// ---- VISUs/Tela_Manual_1.TcVIS
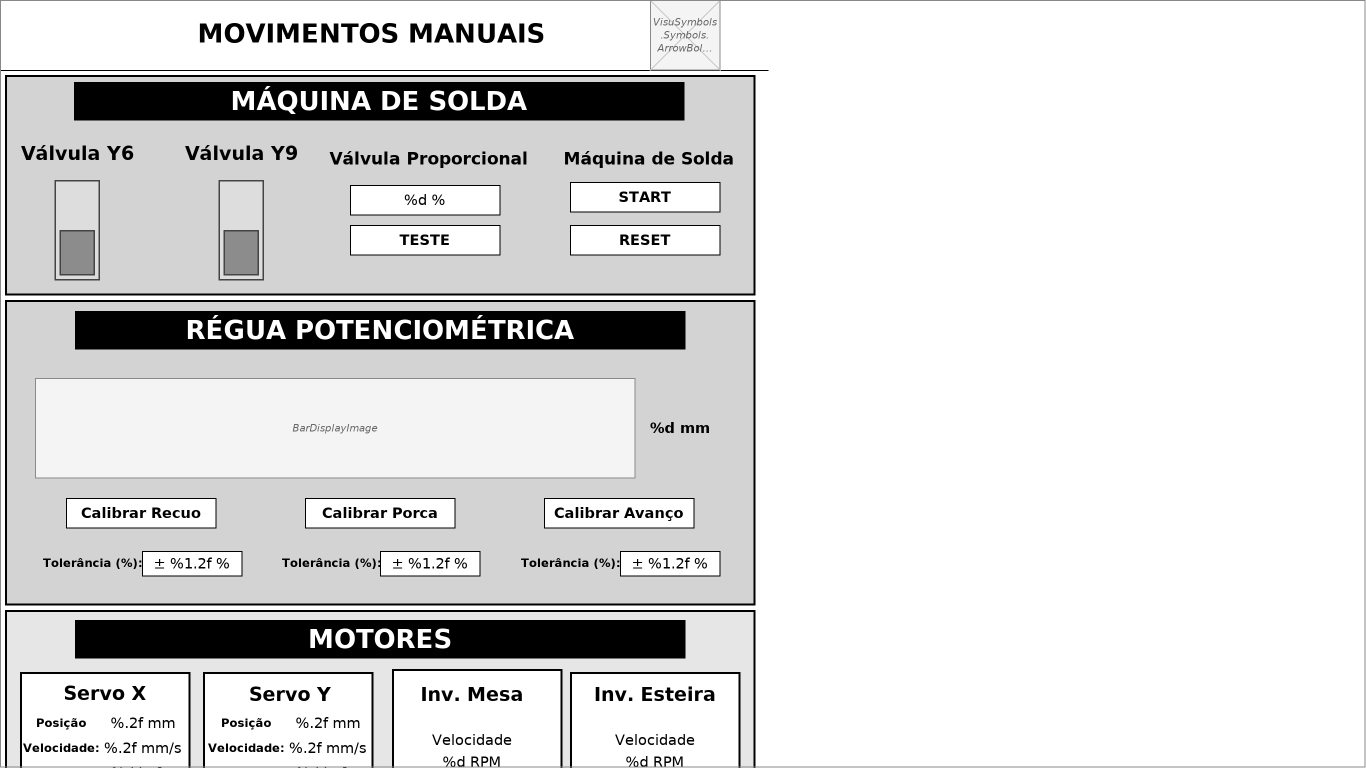
VISUALIZATION Tela_Manual_1  // 1366x768
    Line (0,70) (768,70), input disabled if: NOT MaquinaModoManual
    Line (0,1312) (768,1312)
    Rectangle (584,1340 180x24), "%t[dd/MM/yyyy]"
    Rectangle (584,1316 180x24), "%t[HH:mm:ss]"
    Label (153,7 437x53), "MOVIMENTOS MANUAIS"
    Button (15,1315 175x45), "RECEITAS"
        OnMouseClick: change screen: Tela_Receita
    Button (375,1315 175x45), "MANUTENÇÃO"
        OnMouseClick: change screen: Tela_Manutencao
    RoundedRectangle (5,75 750x220)
    Rectangle (74,82 610x38), "MÁQUINA DE SOLDA", text variable: Recipe_name_Select, input disabled if: NOT MaquinaModoManual
    RoundedRectangle (5,610 750x691), input disabled if: NOT MaquinaModoManual
    Rectangle (75,620 610x38), "MOTORES", text variable: Recipe_name_Select, input disabled if: NOT MaquinaModoManual
    RoundedRectangle (570,672 170x420), input disabled if: NOT MaquinaModoManual
    PushSwitch (625,907 60x60), variable: IhmBt_EsteiraSaida_LigarDesligar, input disabled if: NOT MaquinaModoManual, behaviour: TOGGLE, style: Switch-PushSwitch-Green
    Rectangle (575,681 160x27), "Inv. Esteira", text variable: Recipe_name_Select, input disabled if: NOT MaquinaModoManual
    Rectangle (602,729 106x22), "Velocidade", text variable: Recipe_name_Select, input disabled if: NOT MaquinaModoManual
    Rectangle (602,751 106x22), "%d RPM", text variable: Recipe_name_Select, input disabled if: NOT MaquinaModoManual
    Rectangle (602,879 106x22), "Liga/Desliga", text variable: Recipe_name_Select, input disabled if: NOT MaquinaModoManual
    RotarySwitch (625,803 60x60), variable: IhmBt_EsteiraSaida_Sentido, input disabled if: NOT MaquinaModoManual, behaviour: TOGGLE, style: Switch-RotarySwitch-Gray
    Image (582,823 36x20), input disabled if: NOT MaquinaModoManual, image: VisuSymbols.Symbols.ArrowBoldLeft
    Image (692,823 36x20), input disabled if: NOT MaquinaModoManual, image: VisuSymbols.Symbols.ArrowBoldRight
    RoundedRectangle (392,669 170x420), input disabled if: NOT MaquinaModoManual
    Rectangle (394,681 156x27), "Inv. Mesa", text variable: Recipe_name_Select, input disabled if: NOT MaquinaModoManual
    Rectangle (419,729 106x22), "Velocidade", text variable: Recipe_name_Select, input disabled if: NOT MaquinaModoManual
    Rectangle (419,751 106x22), "%d RPM", text variable: Recipe_name_Select, input disabled if: NOT MaquinaModoManual
    Group (404,803 147x60), input disabled if: NOT MaquinaModoManual
        RotarySwitch (44,0 60x60), variable: IhmBt_MesaIndex_Sentido, behaviour: TOGGLE, style: Switch-RotarySwitch-Gray
        Image (0,20 36x20), image: VisuSymbols.Symbols.ArrowBoldLeft
        Image (111,20 36x20), image: VisuSymbols.Symbols.ArrowBoldRight
    RoundedRectangle (20,672 170x360), input disabled if: NOT MaquinaModoManual
    Rectangle (52,680 106x27), "Servo X", text variable: Recipe_name_Select, input disabled if: NOT MaquinaModoManual
    Rectangle (23,712 77x22), "Posição", input disabled if: NOT MaquinaModoManual
    Rectangle (98,712 90x22), "%.2f mm", text variable: IhmLeit_ServoX_Posicao, input disabled if: NOT MaquinaModoManual
    RoundedRectangle (30,982 150x30), "REFERENCIAR", input disabled if: NOT MaquinaModoManual
        tap IhmBt_ServoX_Referenciar
    RoundedRectangle (30,942 150x30), "POWER ON", input disabled if: NOT MaquinaModoManual
        toggle IhmBt_ServoX_PowerOn
    RoundedRectangle (30,842 150x30), "HOME", colour toggle: NOT Servos.PowerOnServoX, input disabled if: NOT MaquinaModoManual
        tap IhmBt_ServoX_Home
    RoundedRectangle (30,802 150x30), "RESET", input disabled if: NOT MaquinaModoManual
        tap IhmBt_ServoX_Reset
    Image (30,882 50x50), invisible if: NOT IhmBt_ServoX_PowerOn, input disabled if: NOT MaquinaModoManual, image: VisuSymbols.Symbols.ArrowBoldLeft
        OnMouseDown: execute { IhmBt_ServoX_JogBwd := TRUE; }
        OnMouseLeave: execute { IhmBt_ServoX_JogBwd := FALSE; }
        OnMouseUp: execute { IhmBt_ServoX_JogBwd := FALSE; }
    Image (130,882 50x50), invisible if: NOT IhmBt_ServoX_PowerOn, input disabled if: NOT MaquinaModoManual, image: VisuSymbols.Symbols.ArrowBoldRight
        OnMouseDown: execute { IhmBt_ServoX_JogFwd := TRUE; }
        OnMouseLeave: execute { IhmBt_ServoX_JogFwd := FALSE; }
        OnMouseUp: execute { IhmBt_ServoX_JogFwd := FALSE; }
    Rectangle (82,896 45x20), "JOG", invisible if: NOT IhmBt_ServoX_PowerOn, input disabled if: NOT MaquinaModoManual
    Rectangle (23,737 77x22), "Velocidade:", input disabled if: NOT MaquinaModoManual
    Rectangle (98,737 90x22), "%.2f mm/s", text variable: IhmLeit_ServoX_Velocidade, input disabled if: NOT MaquinaModoManual
    Rectangle (23,762 77x22), "Torque:", input disabled if: NOT MaquinaModoManual
    Rectangle (98,762 90x22), "%d kgfm", text variable: IhmLeit_ServoX_Torque, input disabled if: NOT MaquinaModoManual
    RoundedRectangle (203,672 170x360), input disabled if: NOT MaquinaModoManual
    Rectangle (237,681 106x27), "Servo Y", text variable: Recipe_name_Select, input disabled if: NOT MaquinaModoManual
    RoundedRectangle (215,982 150x30), "REFERENCIAR", input disabled if: NOT MaquinaModoManual
        tap IhmBt_ServoY_Referenciar
    RoundedRectangle (215,942 150x30), "POWER ON", input disabled if: NOT MaquinaModoManual
        toggle IhmBt_ServoY_PowerOn
    RoundedRectangle (215,842 150x30), "HOME", colour toggle: NOT Servos.PowerOnServoX, input disabled if: NOT MaquinaModoManual
        tap IhmBt_ServoY_Home
    RoundedRectangle (215,802 150x30), "RESET", input disabled if: NOT MaquinaModoManual
        tap IhmBt_ServoY_Reset
    Image (215,882 50x50), invisible if: NOT IhmBt_ServoY_PowerOn, input disabled if: NOT MaquinaModoManual, image: VisuSymbols.Symbols.ArrowBoldLeft
        OnMouseUp: execute { IhmBt_ServoY_JogBwd := FALSE; }
        OnMouseLeave: execute { IhmBt_ServoY_JogBwd := FALSE; }
        OnMouseDown: execute { IhmBt_ServoY_JogBwd := TRUE; }
    Image (315,882 50x50), invisible if: NOT IhmBt_ServoY_PowerOn, input disabled if: NOT MaquinaModoManual, image: VisuSymbols.Symbols.ArrowBoldRight
        OnMouseUp: execute { IhmBt_ServoY_JogFwd := FALSE; }
        OnMouseLeave: execute { IhmBt_ServoY_JogFwd := FALSE; }
        OnMouseDown: execute { IhmBt_ServoY_JogFwd := TRUE; }
    Rectangle (267,896 45x20), "JOG", text variable: Recipe_name_Select, invisible if: NOT IhmBt_ServoY_PowerOn, input disabled if: NOT MaquinaModoManual
    Rectangle (208,712 77x22), "Posição", input disabled if: NOT MaquinaModoManual
    Rectangle (208,737 77x22), "Velocidade:", input disabled if: NOT MaquinaModoManual
    Rectangle (208,762 77x22), "Torque:", input disabled if: NOT MaquinaModoManual
    Rectangle (283,762 90x22), "%d kgfm", text variable: IhmLeit_ServoY_Torque, input disabled if: NOT MaquinaModoManual
    Rectangle (283,712 90x22), "%.2f mm", text variable: IhmLeit_ServoY_Posicao, input disabled if: NOT MaquinaModoManual
    Rectangle (283,737 90x22), "%.2f mm/s", text variable: IhmLeit_ServoY_Velocidade, input disabled if: NOT MaquinaModoManual
    RoundedRectangle (388,1098 353x125), input disabled if: NOT MaquinaModoManual
    Rectangle (411,1132 130x20), "Frequência (Mesa):", input disabled if: NOT MaquinaModoManual
    Rectangle (584,1132 130x25), "%d Hz", text variable: IhmEscr_MesaIndex_Frequencia, input disabled if: NOT MaquinaModoManual
        OnMouseClick: write the text variable via Default, min 0, max 60
    Rectangle (584,1162 130x25), "%1.2f s", text variable: IhmEscr_MesaIndex_DelayParada, input disabled if: NOT MaquinaModoManual
        OnMouseClick: write the text variable via Default, min 0
    Rectangle (408,1165 130x20), "Delay (Parada)", input disabled if: NOT MaquinaModoManual
    Rectangle (388,1099 353x27), "Ajustes - Inversores", text variable: Recipe_name_Select, input disabled if: NOT MaquinaModoManual
    RoundedRectangle (20,1038 353x185), input disabled if: NOT MaquinaModoManual
    Rectangle (116,1039 160x27), "Ajustes - Servos", text variable: Recipe_name_Select, input disabled if: NOT MaquinaModoManual
    RoundedRectangle (231,1185 50x30), "x100", input disabled if: NOT MaquinaModoManual
        toggle IhmBt_ServoXY_X100
    RoundedRectangle (111,1185 50x30), "x1", input disabled if: NOT MaquinaModoManual
        toggle IhmBt_ServoXY_X1
    RoundedRectangle (171,1185 50x30), "x10", input disabled if: NOT MaquinaModoManual
        toggle IhmBt_ServoXY_X10
    Rectangle (220,1066 130x25), "%d kgf", text variable: IhmEscr_ServoXY_TorqueMax, input disabled if: NOT MaquinaModoManual
        OnMouseClick: write the text variable via Default, min 0, max 300
    Rectangle (44,1069 130x20), "Torque Máximo:", input disabled if: NOT MaquinaModoManual
    Rectangle (220,1095 130x25), "%1.2f s", text variable: IhmEscr_ServoXY_TempoTorqueMax, input disabled if: NOT MaquinaModoManual
        OnMouseClick: write the text variable via Default, min 0, max 300
    Rectangle (43,1098 170x20), "Tempo (Torque Máximo):", input disabled if: NOT MaquinaModoManual
    Rectangle (44,1155 130x20), "Velocidade (Manual):", input disabled if: NOT MaquinaModoManual
    Rectangle (220,1155 130x25), "%d mm/s", text variable: IhmEscr_ServoXY_VelocidadeManual, input disabled if: TRUE
        OnMouseClick: write the text variable via Default, min 0, max 300
    Rectangle (220,1125 130x25), "%d mm/s", text variable: IhmEscr_ServoXY_VelocidadeAuto, input disabled if: NOT MaquinaModoManual
        OnMouseClick: write the text variable via Default, min 0, max 300
    Rectangle (44,1128 130x20), "Velocidade (Auto):", input disabled if: NOT MaquinaModoManual
    Group (404,879 146x192), input disabled if: NOT MaquinaModoManual
        PushSwitch (43,28 60x60), variable: IhmBt_MesaIndex_LigarDesligar, behaviour: TOGGLE, style: Switch-PushSwitch-Green
        Rectangle (20,0 106x22), "Liga/Desliga", text variable: Recipe_name_Select
        PushSwitch (43,132 60x60), variable: IhmBt_MesaIndex_Ciclo, behaviour: TAP, style: Switch-PushSwitch-Green
        Rectangle (0,104 146x22), "Revolução", text variable: Recipe_name_Select
    Image (650,0 70x70), image: VisuSymbols.Symbols.ArrowBoldRight
        OnMouseClick: change screen: Tela_Manual_2
    Image (686,1148 0x1), input disabled if: NOT MaquinaModoManual, image: ImagePool.bt_REFRESH
    Rectangle (584,1192 130x25), "%d Hz", text variable: IhmEscr_EsteiraSaida_Frequencia, input disabled if: NOT MaquinaModoManual
        OnMouseClick: write the text variable via Default, min 0, max 300
    Rectangle (408,1195 130x20), "Frequência (Esteira):", input disabled if: NOT MaquinaModoManual
    Button (195,1315 175x45), "PRODUÇÃO"
        OnMouseClick: change screen: Tela_Producao
    Button (260,1235 240x60), "MODO: %s", text variable: IhmBt_ManualAuto_Text, colour toggle: IhmBt_ManualAuto_Color
        toggle IhmBt_ManualAuto
    Group (20,140 279x140), input disabled if: NOT MaquinaModoManual
        Rectangle (0,0 115x27), "Válvula Y6", text variable: Recipe_name_Select, input disabled if: MaquinaModoAuto
        DipSwitch (7,40 100x100), variable: IhmBt_Y6_Ligar, input disabled if: MaquinaModoAuto, behaviour: TOGGLE, style: Switch-DipSwitch-Gray
        Rectangle (164,0 115x27), "Válvula Y9", text variable: Recipe_name_Select, input disabled if: MaquinaModoAuto
        DipSwitch (171,40 100x100), variable: IhmBt_Y9_Ligar, input disabled if: MaquinaModoAuto, behaviour: TOGGLE, style: Switch-DipSwitch-Gray
    Rectangle (319,145 220x27), "Válvula Proporcional", text variable: Recipe_name_Select, input disabled if: NOT MaquinaModoManual
    RoundedRectangle (350,225 150x30), "TESTE", colour toggle: NOT Servos.PowerOnServoX, input disabled if: NOT MaquinaModoManual
        tap IhmBt_VP_Teste
    Rectangle (350,185 150x30), "%d %", text variable: IhmEscr_ValvulaProporcional, input disabled if: NOT MaquinaModoManual
        OnMouseClick: write the text variable via Default, min 0, max 100
    Rectangle (539,145 220x27), "Máquina de Solda", text variable: Recipe_name_Select, input disabled if: NOT MaquinaModoManual
    RoundedRectangle (570,225 150x30), "RESET", colour toggle: NOT Servos.PowerOnServoX, input disabled if: NOT MaquinaModoManual
        tap IhmBt_MaquinaSolda_Reset
    RoundedRectangle (570,182 150x30), "START", colour toggle: NOT Servos.PowerOnServoX, input disabled if: NOT MaquinaModoManual
        toggle IhmBt_MaquinaSolda_Start
    RoundedRectangle (5,300 750x305)
    Rectangle (75,311 610x38), "RÉGUA POTENCIOMÉTRICA", text variable: Recipe_name_Select, input disabled if: NOT MaquinaModoManual
    Group (35,378 690x198)
        RoundedRectangle (31,120 150x30), "Calibrar Recuo", input disabled if: NOT MaquinaModoManual
            tap IhmBt_ReguaPotenciometrica_CalibrarRecuo
        Rectangle (5,175 100x20), "Tolerância (%):", input disabled if: NOT MaquinaModoManual
        BarDisplayImage (0,0 600x100), value: ReguaPotenciometricaPosicao, style: BarDisplayImage-Gray, scale format: %.1f, scale 0..100
            p518627256: mm
        Rectangle (600,39 90x22), "%d mm", text variable: ReguaPotenciometricaPosicao, input disabled if: TRUE
        Rectangle (244,175 100x20), "Tolerância (%):", input disabled if: NOT MaquinaModoManual
        RoundedRectangle (270,120 150x30), "Calibrar Porca", input disabled if: NOT MaquinaModoManual
            tap IhmBt_ReguaPotenciometrica_CalibrarPorca
        RoundedRectangle (509,120 150x30), "Calibrar Avanço", input disabled if: NOT MaquinaModoManual
            tap IhmBt_ReguaPotenciometrica_CalibrarAvanco
        Rectangle (483,175 100x20), "Tolerância (%):", input disabled if: NOT MaquinaModoManual
        Rectangle (107,173 100x25), "± %1.2f %", text variable: IhmEscr_ReguaPotenciometrica_ToleranciaRecuo, input disabled if: NOT MaquinaModoManual
            OnMouseClick: write the text variable via Default, min 0, max 100
        Rectangle (345,173 100x25), "± %1.2f %", text variable: IhmEscr_ReguaPotenciometrica_ToleranciaPorca, input disabled if: NOT MaquinaModoManual
            OnMouseClick: write the text variable via Default, min 0, max 100
        Rectangle (585,173 100x25), "± %1.2f %", text variable: IhmEscr_ReguaPotenciometrica_ToleranciaAvanco, input disabled if: NOT MaquinaModoManual
            OnMouseClick: write the text variable via Default, min 0, max 100
END_VISUALIZATION

// ---- VISUs/Tela_Receita.TcVIS
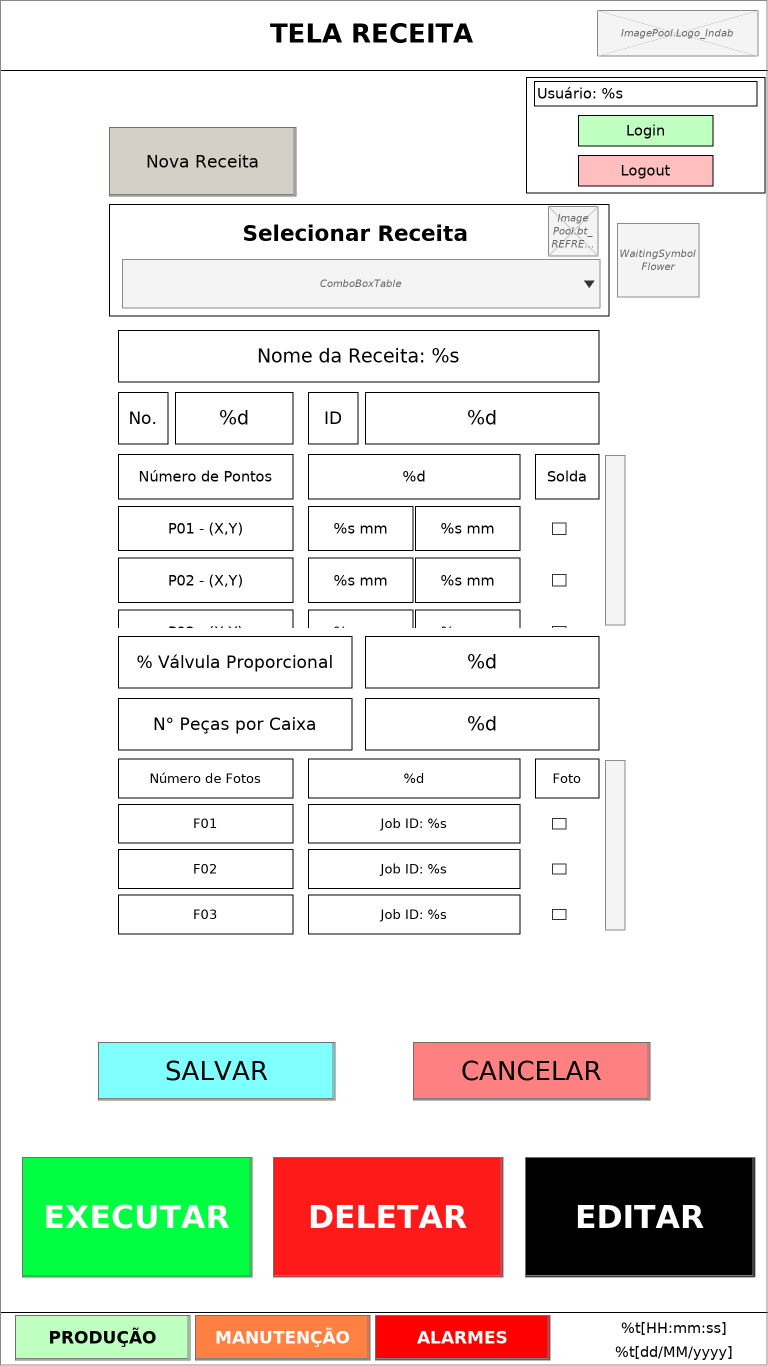
VISUALIZATION Tela_Receita  // 768x1366, background image __VisualizationStyle.CheckboxChecked
    Frame (113,450 492x675)
        shows Lista_PontosSolda()
        shows Lista_PontosRoboCamera()
        p2738717112: Main_Receita.ScrollScreen_PontosSolda
    Rectangle (-1,628 768x500)
    Rectangle (-1,628 768x737)
    Frame (113,755 492x275)
        shows Lista_PontosRoboCamera()
        shows Lista_PontosRoboCamera()
        p2738717112: Main_Receita.ScrollScreen_PontosSolda
    Rectangle (-1,0 768x450)
    Rectangle (109,204 500x112)
    Line (0,70) (768,70)
    Image (597,10 161x46), image: ImagePool.Logo_Indab
    Label (153,7 437x53), "TELA RECEITA"
    ComboBoxTable (122,259 478x49), variable: Recipe_select_int, input disabled if: b_editar_receita or b_criar_receita, data array: Recipe_names_saved
        p1128707560: Main_Receita.Item_livre
        p3854506369: Recipe_names_saved[INDEX]
    Rectangle (118,330 481x52), "Nome da Receita: %s", text variable: Recipe_name_Select, input disabled if: Not b_editar_receita and Not b_criar_receita
        OnMouseClick: write the text variable via Default
    Rectangle (526,77 239x116)
    Rectangle (578,115 135x31), "Login"
        OnMouseClick: VisuUserMgmt Type=Login
    Rectangle (578,155 135x31), "Logout"
        OnMouseClick: VisuUserMgmt Type=Logout
    Rectangle (534,81 223x25), "Usuário: %s", text variable: UserName
    Button (109,127 187x69), "Nova Receita"
        OnMouseClick: execute { b_criar_receita := TRUE; }
    Label (137,207 437x53), "Selecionar Receita"
    WaitingSymbolFlower (617,223 82x74), invisible if: Not Simbolo_Atualizacao
    Image (548,206 50x50), image: ImagePool.bt_REFRESH
        OnMouseClick: execute { bRead := TRUE; }
    Scrollbar (605,455 20x170), invisible if: Recipe_Pontos_Solda_Select<=3
        p2245068023: Main_Receita.LengthScrollBar_PontosSolda
        p1057716461: Main_Receita.ScrollBar_PontosSolda
    Rectangle (365,392 234x52), "%d", text variable: Recipe_ID_Select, input disabled if: Not b_editar_receita and Not b_criar_receita
        OnMouseClick: write the text variable via Default
    Rectangle (118,392 50x52), "No."
    Rectangle (175,392 118x52), "%d", text variable: Recipe_No_Select, input disabled if: Not b_editar_receita and Not b_criar_receita
        OnMouseClick: write the text variable via Default
    Rectangle (308,392 50x52), "ID"
    Scrollbar (605,760 20x170), invisible if: Recipe_Pontos_Camera_Select<=3
        p2245068023: Main_Receita.LengthScrollBar_PontosCamera
        p1057716461: Main_Receita.ScrollBar_PontosCamera
    Rectangle (-1,630 768x125)
    Rectangle (118,636 234x52), "% Válvula Proporcional"
    Rectangle (365,636 234x52), "%d", text variable: Recipe_Valvula_Proporcional_Select, input disabled if: Not b_editar_receita and Not b_criar_receita
        OnMouseClick: write the text variable via Default
    Rectangle (365,698 234x52), "%d", text variable: Recipe_Pecas_Caixa_Select, input disabled if: Not b_editar_receita and Not b_criar_receita
        OnMouseClick: write the text variable via Default
    Rectangle (118,698 234x52), "N° Peças por Caixa"
    Line (0,1312) (768,1312)
    Rectangle (584,1340 180x24), "%t[dd/MM/yyyy]"
    Rectangle (584,1316 180x24), "%t[HH:mm:ss]"
    Rectangle (-1,940 768x365)
    Button (525,1157 230x120), "EDITAR", input disabled if: b_criar_receita
        OnMouseClick: execute { b_editar_receita := TRUE; }
    Button (22,1157 230x120), "EXECUTAR", input disabled if: b_editar_receita
        OnMouseClick: execute { b_executar_receita := TRUE; }
    Button (273,1157 230x120), "DELETAR", input disabled if: Not b_editar_receita
        OnMouseClick: execute { b_deletar_receita := TRUE; }
    Button (98,1042 237x58), "SALVAR", invisible if: Not b_editar_receita AND Not b_criar_receita
        OnMouseClick: execute { b_salvar_receita := TRUE; }
    Button (413,1042 237x58), "CANCELAR", invisible if: Not b_editar_receita AND NOT b_criar_receita
        OnMouseClick: execute { b_cancelar_receita := TRUE; }
    Button (15,1315 175x45), "PRODUÇÃO"
        OnMouseClick: change screen: Tela_Producao
    Button (195,1315 175x45), "MANUTENÇÃO"
        OnMouseClick: change screen: Tela_Manutencao
    Button (375,1315 175x45), "ALARMES"
        OnMouseClick: change screen: Tela_Alarmes_1
END_VISUALIZATION

// ---- VISUs/Tela_Manutencao.TcVIS
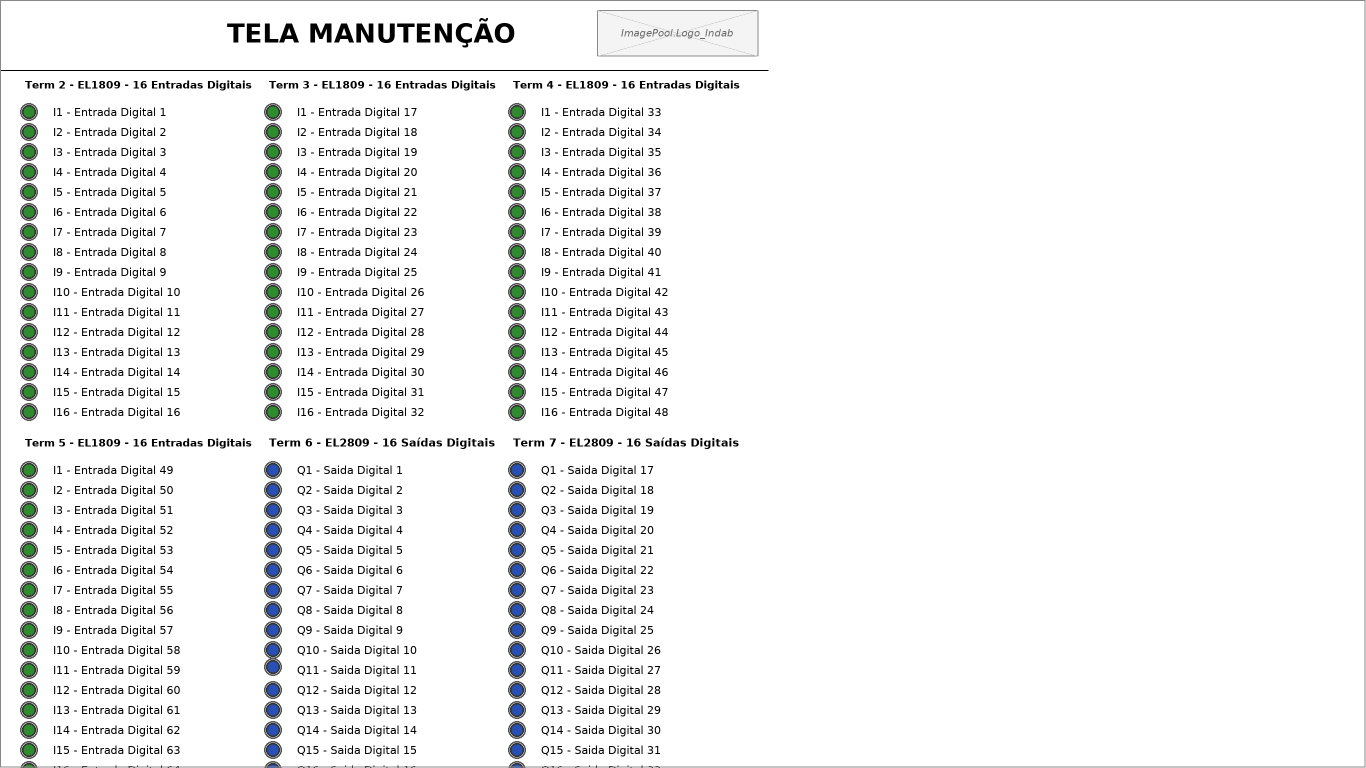
VISUALIZATION Tela_Manutencao  // 1366x768
    Line (0,70) (768,70)
    Line (0,1312) (768,1312)
    Image (597,10 161x46), image: ImagePool.Logo_Indab
    Rectangle (584,1340 180x24), "%t[dd/MM/yyyy]"
    Rectangle (584,1316 180x24), "%t[HH:mm:ss]"
    Label (153,7 437x53), "TELA MANUTENÇÃO"
    Group (19,75 244x347)
        Lamp1 (0,27 20x20), variable: EntradaI0_0, style: Lamp-Lamp1-Green
        Rectangle (31,28 213x19), "I1 - Entrada Digital 1"
        Lamp1 (0,47 20x20), variable: EntradaI0_1, style: Lamp-Lamp1-Green
        Rectangle (31,48 213x19), "I2 - Entrada Digital 2"
        Lamp1 (0,67 20x20), variable: EntradaI0_2, style: Lamp-Lamp1-Green
        Rectangle (31,68 213x19), "I3 - Entrada Digital 3"
        Lamp1 (0,87 20x20), variable: EntradaI0_3, style: Lamp-Lamp1-Green
        Rectangle (31,88 213x19), "I4 - Entrada Digital 4"
        Lamp1 (0,107 20x20), variable: EntradaI0_4, style: Lamp-Lamp1-Green
        Rectangle (31,108 213x19), "I5 - Entrada Digital 5"
        Lamp1 (0,127 20x20), variable: EntradaI0_5, style: Lamp-Lamp1-Green
        Rectangle (31,128 213x19), "I6 - Entrada Digital 6"
        Lamp1 (0,147 20x20), variable: EntradaI0_6, style: Lamp-Lamp1-Green
        Rectangle (31,148 213x19), "I7 - Entrada Digital 7"
        Lamp1 (0,167 20x20), variable: EntradaI0_7, style: Lamp-Lamp1-Green
        Rectangle (31,168 213x19), "I8 - Entrada Digital 8"
        Lamp1 (0,187 20x20), variable: EntradaI1_0, style: Lamp-Lamp1-Green
        Rectangle (31,188 213x19), "I9 - Entrada Digital 9"
        Lamp1 (0,207 20x20), variable: EntradaI1_1, style: Lamp-Lamp1-Green
        Rectangle (31,208 213x19), "I10 - Entrada Digital 10"
        Lamp1 (0,227 20x20), variable: EntradaI1_2, style: Lamp-Lamp1-Green
        Rectangle (31,228 213x19), "I11 - Entrada Digital 11"
        Lamp1 (0,247 20x20), variable: EntradaI1_3, style: Lamp-Lamp1-Green
        Rectangle (31,248 213x19), "I12 - Entrada Digital 12"
        Lamp1 (0,267 20x20), variable: EntradaI1_4, style: Lamp-Lamp1-Green
        Rectangle (31,268 213x19), "I13 - Entrada Digital 13"
        Lamp1 (0,287 20x20), variable: EntradaI1_5, style: Lamp-Lamp1-Green
        Rectangle (31,288 213x19), "I14 - Entrada Digital 14"
        Lamp1 (0,307 20x20), variable: EntradaI1_6, style: Lamp-Lamp1-Green
        Rectangle (31,308 213x19), "I15 - Entrada Digital 15"
        Lamp1 (0,327 20x20), variable: EntradaI1_7, style: Lamp-Lamp1-Green
        Rectangle (31,328 213x19), "I16 - Entrada Digital 16"
        Rectangle (3,0 237x20), "Term 2 - EL1809 - 16 Entradas Digitais"
    Group (19,433 244x347)
        Lamp1 (0,27 20x20), variable: EntradaI6_0, style: Lamp-Lamp1-Green
        Rectangle (31,28 213x19), "I1 - Entrada Digital 49"
        Lamp1 (0,47 20x20), variable: EntradaI6_1, style: Lamp-Lamp1-Green
        Rectangle (31,48 213x19), "I2 - Entrada Digital 50"
        Lamp1 (0,67 20x20), variable: EntradaI6_2, style: Lamp-Lamp1-Green
        Rectangle (31,68 213x19), "I3 - Entrada Digital 51"
        Lamp1 (0,87 20x20), variable: EntradaI6_3, style: Lamp-Lamp1-Green
        Rectangle (31,88 213x19), "I4 - Entrada Digital 52"
        Lamp1 (0,107 20x20), variable: EntradaI6_4, style: Lamp-Lamp1-Green
        Rectangle (31,108 213x19), "I5 - Entrada Digital 53"
        Lamp1 (0,127 20x20), variable: EntradaI6_5, style: Lamp-Lamp1-Green
        Rectangle (31,128 213x19), "I6 - Entrada Digital 54"
        Lamp1 (0,147 20x20), variable: EntradaI6_6, style: Lamp-Lamp1-Green
        Rectangle (31,148 213x19), "I7 - Entrada Digital 55"
        Lamp1 (0,167 20x20), variable: EntradaI6_7, style: Lamp-Lamp1-Green
        Rectangle (31,168 213x19), "I8 - Entrada Digital 56"
        Lamp1 (0,187 20x20), variable: EntradaI7_0, style: Lamp-Lamp1-Green
        Rectangle (31,188 213x19), "I9 - Entrada Digital 57"
        Lamp1 (0,207 20x20), variable: EntradaI7_1, style: Lamp-Lamp1-Green
        Rectangle (31,208 213x19), "I10 - Entrada Digital 58"
        Lamp1 (0,227 20x20), variable: EntradaI7_2, style: Lamp-Lamp1-Green
        Rectangle (31,228 213x19), "I11 - Entrada Digital 59"
        Lamp1 (0,247 20x20), variable: EntradaI7_3, style: Lamp-Lamp1-Green
        Rectangle (31,248 213x19), "I12 - Entrada Digital 60"
        Lamp1 (0,267 20x20), variable: EntradaI7_4, style: Lamp-Lamp1-Green
        Rectangle (31,268 213x19), "I13 - Entrada Digital 61"
        Lamp1 (0,287 20x20), variable: EntradaI7_5, style: Lamp-Lamp1-Green
        Rectangle (31,288 213x19), "I14 - Entrada Digital 62"
        Lamp1 (0,307 20x20), variable: EntradaI7_6, style: Lamp-Lamp1-Green
        Rectangle (31,308 213x19), "I15 - Entrada Digital 63"
        Lamp1 (0,327 20x20), variable: EntradaI7_7, style: Lamp-Lamp1-Green
        Rectangle (31,328 213x19), "I16 - Entrada Digital 64"
        Rectangle (3,0 237x20), "Term 5 - EL1809 - 16 Entradas Digitais"
    Group (263,75 244x347)
        Lamp1 (0,27 20x20), variable: EntradaI2_0, style: Lamp-Lamp1-Green
        Rectangle (31,28 213x19), "I1 - Entrada Digital 17"
        Lamp1 (0,47 20x20), variable: EntradaI2_1, style: Lamp-Lamp1-Green
        Rectangle (31,48 213x19), "I2 - Entrada Digital 18"
        Lamp1 (0,67 20x20), variable: EntradaI2_2, style: Lamp-Lamp1-Green
        Rectangle (31,68 213x19), "I3 - Entrada Digital 19"
        Lamp1 (0,87 20x20), variable: EntradaI2_3, style: Lamp-Lamp1-Green
        Rectangle (31,88 213x19), "I4 - Entrada Digital 20"
        Lamp1 (0,107 20x20), variable: EntradaI2_4, style: Lamp-Lamp1-Green
        Rectangle (31,108 213x19), "I5 - Entrada Digital 21"
        Lamp1 (0,127 20x20), variable: EntradaI2_5, style: Lamp-Lamp1-Green
        Rectangle (31,128 213x19), "I6 - Entrada Digital 22"
        Lamp1 (0,147 20x20), variable: EntradaI2_6, style: Lamp-Lamp1-Green
        Rectangle (31,148 213x19), "I7 - Entrada Digital 23"
        Lamp1 (0,167 20x20), variable: EntradaI2_7, style: Lamp-Lamp1-Green
        Rectangle (31,168 213x19), "I8 - Entrada Digital 24"
        Lamp1 (0,187 20x20), variable: EntradaI3_0, style: Lamp-Lamp1-Green
        Rectangle (31,188 213x19), "I9 - Entrada Digital 25"
        Lamp1 (0,207 20x20), variable: EntradaI3_1, style: Lamp-Lamp1-Green
        Rectangle (31,208 213x19), "I10 - Entrada Digital 26"
        Lamp1 (0,227 20x20), variable: EntradaI3_2, style: Lamp-Lamp1-Green
        Rectangle (31,228 213x19), "I11 - Entrada Digital 27"
        Lamp1 (0,247 20x20), variable: EntradaI3_3, style: Lamp-Lamp1-Green
        Rectangle (31,248 213x19), "I12 - Entrada Digital 28"
        Lamp1 (0,267 20x20), variable: EntradaI3_4, style: Lamp-Lamp1-Green
        Rectangle (31,268 213x19), "I13 - Entrada Digital 29"
        Lamp1 (0,287 20x20), variable: EntradaI3_5, style: Lamp-Lamp1-Green
        Rectangle (31,288 213x19), "I14 - Entrada Digital 30"
        Lamp1 (0,307 20x20), variable: EntradaI3_6, style: Lamp-Lamp1-Green
        Rectangle (31,308 213x19), "I15 - Entrada Digital 31"
        Lamp1 (0,327 20x20), variable: EntradaI3_7, style: Lamp-Lamp1-Green
        Rectangle (31,328 213x19), "I16 - Entrada Digital 32"
        Rectangle (3,0 239x20), "Term 3 - EL1809 - 16 Entradas Digitais"
    Group (507,75 244x347)
        Lamp1 (0,27 20x20), variable: EntradaI4_0, style: Lamp-Lamp1-Green
        Rectangle (31,28 213x19), "I1 - Entrada Digital 33"
        Lamp1 (0,47 20x20), variable: EntradaI4_1, style: Lamp-Lamp1-Green
        Rectangle (31,48 213x19), "I2 - Entrada Digital 34"
        Lamp1 (0,67 20x20), variable: EntradaI4_2, style: Lamp-Lamp1-Green
        Rectangle (31,68 213x19), "I3 - Entrada Digital 35"
        Lamp1 (0,87 20x20), variable: EntradaI4_3, style: Lamp-Lamp1-Green
        Rectangle (31,88 213x19), "I4 - Entrada Digital 36"
        Lamp1 (0,107 20x20), variable: EntradaI4_4, style: Lamp-Lamp1-Green
        Rectangle (31,108 213x19), "I5 - Entrada Digital 37"
        Lamp1 (0,127 20x20), variable: EntradaI4_5, style: Lamp-Lamp1-Green
        Rectangle (31,128 213x19), "I6 - Entrada Digital 38"
        Lamp1 (0,147 20x20), variable: EntradaI4_6, style: Lamp-Lamp1-Green
        Rectangle (31,148 213x19), "I7 - Entrada Digital 39"
        Lamp1 (0,167 20x20), variable: EntradaI4_7, style: Lamp-Lamp1-Green
        Rectangle (31,168 213x19), "I8 - Entrada Digital 40"
        Lamp1 (0,187 20x20), variable: EntradaI5_0, style: Lamp-Lamp1-Green
        Rectangle (31,188 213x19), "I9 - Entrada Digital 41"
        Lamp1 (0,207 20x20), variable: EntradaI5_1, style: Lamp-Lamp1-Green
        Rectangle (31,208 213x19), "I10 - Entrada Digital 42"
        Lamp1 (0,227 20x20), variable: EntradaI5_2, style: Lamp-Lamp1-Green
        Rectangle (31,228 213x19), "I11 - Entrada Digital 43"
        Lamp1 (0,247 20x20), variable: EntradaI5_3, style: Lamp-Lamp1-Green
        Rectangle (31,248 213x19), "I12 - Entrada Digital 44"
        Lamp1 (0,267 20x20), variable: EntradaI5_4, style: Lamp-Lamp1-Green
        Rectangle (31,268 213x19), "I13 - Entrada Digital 45"
        Lamp1 (0,287 20x20), variable: EntradaI5_5, style: Lamp-Lamp1-Green
        Rectangle (31,288 213x19), "I14 - Entrada Digital 46"
        Lamp1 (0,307 20x20), variable: EntradaI5_6, style: Lamp-Lamp1-Green
        Rectangle (31,308 213x19), "I15 - Entrada Digital 47"
        Lamp1 (0,327 20x20), variable: EntradaI5_7, style: Lamp-Lamp1-Green
        Rectangle (31,328 213x19), "I16 - Entrada Digital 48"
        Rectangle (3,0 237x20), "Term 4 - EL1809 - 16 Entradas Digitais"
    Group (263,433 244x347)
        Lamp1 (0,27 20x20), variable: SaidaQ0_0, style: Lamp-Lamp1-Blue
        Rectangle (31,28 213x19), "Q1 - Saida Digital 1"
        Lamp1 (0,47 20x20), variable: SaidaQ0_1, style: Lamp-Lamp1-Blue
        Rectangle (31,48 213x19), "Q2 - Saida Digital 2"
        Lamp1 (0,67 20x20), variable: SaidaQ0_2, style: Lamp-Lamp1-Blue
        Rectangle (31,68 213x19), "Q3 - Saida Digital 3"
        Lamp1 (0,87 20x20), variable: SaidaQ0_3, style: Lamp-Lamp1-Blue
        Rectangle (31,88 213x19), "Q4 - Saida Digital 4"
        Lamp1 (0,107 20x20), variable: SaidaQ0_4, style: Lamp-Lamp1-Blue
        Rectangle (31,108 213x19), "Q5 - Saida Digital 5"
        Lamp1 (0,127 20x20), variable: SaidaQ0_5, style: Lamp-Lamp1-Blue
        Rectangle (31,128 213x19), "Q6 - Saida Digital 6"
        Lamp1 (0,147 20x20), variable: SaidaQ0_6, style: Lamp-Lamp1-Blue
        Rectangle (31,148 213x19), "Q7 - Saida Digital 7"
        Lamp1 (0,167 20x20), variable: SaidaQ0_7, style: Lamp-Lamp1-Blue
        Rectangle (31,168 213x19), "Q8 - Saida Digital 8"
        Lamp1 (0,187 20x20), variable: SaidaQ1_0, style: Lamp-Lamp1-Blue
        Rectangle (31,188 213x19), "Q9 - Saida Digital 9"
        Lamp1 (0,207 20x20), variable: SaidaQ1_1, style: Lamp-Lamp1-Blue
        Rectangle (31,208 213x19), "Q10 - Saida Digital 10"
        Lamp1 (0,224 20x20), variable: SaidaQ1_2, style: Lamp-Lamp1-Blue
        Rectangle (31,228 213x19), "Q11 - Saida Digital 11"
        Lamp1 (0,247 20x20), variable: SaidaQ1_3, style: Lamp-Lamp1-Blue
        Rectangle (31,248 213x19), "Q12 - Saida Digital 12"
        Lamp1 (0,267 20x20), variable: SaidaQ1_4, style: Lamp-Lamp1-Blue
        Rectangle (31,268 213x19), "Q13 - Saida Digital 13"
        Lamp1 (0,287 20x20), variable: SaidaQ1_5, style: Lamp-Lamp1-Blue
        Rectangle (31,288 213x19), "Q14 - Saida Digital 14"
        Lamp1 (0,307 20x20), variable: SaidaQ1_6, style: Lamp-Lamp1-Blue
        Rectangle (31,308 213x19), "Q15 - Saida Digital 15"
        Lamp1 (0,327 20x20), variable: SaidaQ1_7, style: Lamp-Lamp1-Blue
        Rectangle (31,328 213x19), "Q16 - Saida Digital 16"
        Rectangle (3,0 237x20), "Term 6 - EL2809 - 16 Saídas Digitais"
    Group (507,433 244x347)
        Lamp1 (0,27 20x20), variable: SaidaQ2_0, style: Lamp-Lamp1-Blue
        Rectangle (31,28 213x19), "Q1 - Saida Digital 17"
        Lamp1 (0,47 20x20), variable: SaidaQ2_1, style: Lamp-Lamp1-Blue
        Rectangle (31,48 213x19), "Q2 - Saida Digital 18"
        Lamp1 (0,67 20x20), variable: SaidaQ2_2, style: Lamp-Lamp1-Blue
        Rectangle (31,68 213x19), "Q3 - Saida Digital 19"
        Lamp1 (0,87 20x20), variable: SaidaQ2_3, style: Lamp-Lamp1-Blue
        Rectangle (31,88 213x19), "Q4 - Saida Digital 20"
        Lamp1 (0,107 20x20), variable: SaidaQ2_4, style: Lamp-Lamp1-Blue
        Rectangle (31,108 213x19), "Q5 - Saida Digital 21"
        Lamp1 (0,127 20x20), variable: SaidaQ2_5, style: Lamp-Lamp1-Blue
        Rectangle (31,128 213x19), "Q6 - Saida Digital 22"
        Lamp1 (0,147 20x20), variable: SaidaQ2_6, style: Lamp-Lamp1-Blue
        Rectangle (31,148 213x19), "Q7 - Saida Digital 23"
        Lamp1 (0,167 20x20), variable: SaidaQ2_7, style: Lamp-Lamp1-Blue
        Rectangle (31,168 213x19), "Q8 - Saida Digital 24"
        Lamp1 (0,187 20x20), variable: SaidaQ3_0, style: Lamp-Lamp1-Blue
        Rectangle (31,188 213x19), "Q9 - Saida Digital 25"
        Lamp1 (0,207 20x20), variable: SaidaQ3_1, style: Lamp-Lamp1-Blue
        Rectangle (31,208 213x19), "Q10 - Saida Digital 26"
        Lamp1 (0,227 20x20), variable: SaidaQ3_2, style: Lamp-Lamp1-Blue
        Rectangle (31,228 213x19), "Q11 - Saida Digital 27"
        Lamp1 (0,247 20x20), variable: SaidaQ3_3, style: Lamp-Lamp1-Blue
        Rectangle (31,248 213x19), "Q12 - Saida Digital 28"
        Lamp1 (0,267 20x20), variable: SaidaQ3_4, style: Lamp-Lamp1-Blue
        Rectangle (31,268 213x19), "Q13 - Saida Digital 29"
        Lamp1 (0,287 20x20), variable: SaidaQ3_5, style: Lamp-Lamp1-Blue
        Rectangle (31,288 213x19), "Q14 - Saida Digital 30"
        Lamp1 (0,307 20x20), variable: SaidaQ3_6, style: Lamp-Lamp1-Blue
        Rectangle (31,308 213x19), "Q15 - Saida Digital 31"
        Lamp1 (0,327 20x20), variable: SaidaQ3_7, style: Lamp-Lamp1-Blue
        Rectangle (31,328 213x19), "Q16 - Saida Digital 32"
        Rectangle (3,0 237x20), "Term 7 - EL2809 - 16 Saídas Digitais"
    Group (19,791 244x347)
        Lamp1 (0,27 20x20), variable: SaidaQ4_0, style: Lamp-Lamp1-Blue
        Rectangle (31,28 213x19), "Q1 - Saida Digital 33"
        Lamp1 (0,47 20x20), variable: SaidaQ4_1, style: Lamp-Lamp1-Blue
        Rectangle (31,48 213x19), "Q2 - Saida Digital 34"
        Lamp1 (0,67 20x20), variable: SaidaQ4_2, style: Lamp-Lamp1-Blue
        Rectangle (31,68 213x19), "Q3 - Saida Digital 35"
        Lamp1 (0,87 20x20), variable: SaidaQ4_3, style: Lamp-Lamp1-Blue
        Rectangle (31,88 213x19), "Q4 - Saida Digital 36"
        Lamp1 (0,107 20x20), variable: SaidaQ4_4, style: Lamp-Lamp1-Blue
        Rectangle (31,108 213x19), "Q5 - Saida Digital 37"
        Lamp1 (0,127 20x20), variable: SaidaQ4_5, style: Lamp-Lamp1-Blue
        Rectangle (31,128 213x19), "Q6 - Saida Digital 38"
        Lamp1 (0,147 20x20), variable: SaidaQ4_6, style: Lamp-Lamp1-Blue
        Rectangle (31,148 213x19), "Q7 - Saida Digital 39"
        Lamp1 (0,167 20x20), variable: SaidaQ4_7, style: Lamp-Lamp1-Blue
        Rectangle (31,168 213x19), "Q8 - Saida Digital 40"
        Lamp1 (0,187 20x20), variable: SaidaQ5_0, style: Lamp-Lamp1-Blue
        Rectangle (31,188 213x19), "Q9 - Saida Digital 41"
        Lamp1 (0,207 20x20), variable: SaidaQ5_1, style: Lamp-Lamp1-Blue
        Rectangle (31,208 213x19), "Q10 - Saida Digital 42"
        Lamp1 (0,227 20x20), variable: SaidaQ5_2, style: Lamp-Lamp1-Blue
        Rectangle (31,228 213x19), "Q11 - Saida Digital 43"
        Lamp1 (0,247 20x20), variable: SaidaQ5_3, style: Lamp-Lamp1-Blue
        Rectangle (31,248 213x19), "Q12 - Saida Digital 44"
        Lamp1 (0,267 20x20), variable: SaidaQ5_4, style: Lamp-Lamp1-Blue
        Rectangle (31,268 213x19), "Q13 - Saida Digital 45"
        Lamp1 (0,287 20x20), variable: SaidaQ5_5, style: Lamp-Lamp1-Blue
        Rectangle (31,288 213x19), "Q14 - Saida Digital 46"
        Lamp1 (0,307 20x20), variable: SaidaQ5_6, style: Lamp-Lamp1-Blue
        Rectangle (31,308 213x19), "Q15 - Saida Digital 47"
        Lamp1 (0,327 20x20), variable: SaidaQ5_7, style: Lamp-Lamp1-Blue
        Rectangle (31,328 213x19), "Q16 - Saida Digital 48"
        Rectangle (3,0 237x20), "Term 8 - EL2809 - 16 Saídas Digitais"
    Group (263,791 244x347)
        Lamp1 (0,27 20x20), variable: SaidaQ6_0, style: Lamp-Lamp1-Blue
        Rectangle (31,28 213x19), "Q1 - Saida Digital 49"
        Lamp1 (0,47 20x20), variable: SaidaQ6_1, style: Lamp-Lamp1-Blue
        Rectangle (31,48 213x19), "Q2 - Saida Digital 50"
        Lamp1 (0,67 20x20), variable: SaidaQ6_2, style: Lamp-Lamp1-Blue
        Rectangle (31,68 213x19), "Q3 - Saida Digital 51"
        Lamp1 (0,87 20x20), variable: SaidaQ6_3, style: Lamp-Lamp1-Blue
        Rectangle (31,88 213x19), "Q4 - Saida Digital 52"
        Lamp1 (0,107 20x20), variable: SaidaQ6_4, style: Lamp-Lamp1-Blue
        Rectangle (31,108 213x19), "Q5 - Saida Digital 53"
        Lamp1 (0,127 20x20), variable: SaidaQ6_5, style: Lamp-Lamp1-Blue
        Rectangle (31,128 213x19), "Q6 - Saida Digital 54"
        Lamp1 (0,147 20x20), variable: SaidaQ6_7, style: Lamp-Lamp1-Blue
        Rectangle (31,148 213x19), "Q7 - Saida Digital 55"
        Lamp1 (0,167 20x20), variable: SaidaQ7_0, style: Lamp-Lamp1-Blue
        Rectangle (31,168 213x19), "Q8 - Saida Digital 56"
        Lamp1 (0,187 20x20), variable: SaidaQ7_1, style: Lamp-Lamp1-Blue
        Rectangle (31,188 213x19), "Q9 - Saida Digital 57"
        Lamp1 (0,207 20x20), variable: SaidaQ7_1, style: Lamp-Lamp1-Blue
        Rectangle (31,208 213x19), "Q10 - Saida Digital 58"
        Lamp1 (0,227 20x20), variable: SaidaQ7_2, style: Lamp-Lamp1-Blue
        Rectangle (31,228 213x19), "Q11 - Saida Digital 59"
        Lamp1 (0,247 20x20), variable: SaidaQ7_3, style: Lamp-Lamp1-Blue
        Rectangle (31,248 213x19), "Q12 - Saida Digital 60"
        Lamp1 (0,267 20x20), variable: SaidaQ7_4, style: Lamp-Lamp1-Blue
        Rectangle (31,268 213x19), "Q13 - Saida Digital 61"
        Lamp1 (0,287 20x20), variable: SaidaQ7_5, style: Lamp-Lamp1-Blue
        Rectangle (31,288 213x19), "Q14 - Saida Digital 62"
        Lamp1 (0,307 20x20), variable: SaidaQ7_6, style: Lamp-Lamp1-Blue
        Rectangle (31,308 213x19), "Q15 - Saida Digital 63"
        Lamp1 (0,327 20x20), variable: SaidaQ7_7, style: Lamp-Lamp1-Blue
        Rectangle (31,328 213x19), "Q16 - Saida Digital 64"
        Rectangle (3,0 237x20), "Term 9 - EL2809 - 16 Saídas Digitais"
    Group (263,1242 244x67)
        Lamp1 (0,27 20x20), variable: I2, style: Lamp-Lamp1-Yellow
        Rectangle (31,28 213x19), "I1 - Entrada Rapida 1"
        Lamp1 (0,47 20x20), variable: I2, style: Lamp-Lamp1-Yellow
        Rectangle (31,48 213x19), "I2 - Entrada Rapida 2"
        Rectangle (3,0 237x20), "Term 9 - EL1252 - 2 Entradas Rápidas"
    Group (19,1146 244x104)
        Rectangle (0,0 237x20), "Term 9 - EL4004 - 4 Saídas Analógicas"
        Group (51,28 202x76)
            Rectangle (0,0 213x19), "AO1 - Saida Analogica 1"
            Rectangle (0,19 213x19), "AO1 - Saida Analogica 2"
            Rectangle (0,38 213x19), "AO1 - Saida Analogica 3"
            Rectangle (0,57 213x19), "AO1 - Saida Analogica 4"
        Group (0,28 51x76)
            Rectangle (0,0 51x19), "%s"
            Rectangle (0,19 51x19), "%s"
            Rectangle (0,38 51x19), "%s"
            Rectangle (0,57 51x19), "%s"
    Group (263,1146 244x87)
        Lamp1 (0,27 20x20), variable: I2, style: Lamp-Lamp1-Yellow
        Rectangle (31,28 213x19), "Robo Yaskawa GP7"
        Lamp1 (0,47 20x20), variable: I2, style: Lamp-Lamp1-Yellow
        Rectangle (31,48 213x19), "Camera Sick Inspector"
        Rectangle (3,0 237x20), "Conexão Ethernet/IP"
        Lamp1 (0,67 20x20), variable: I2, style: Lamp-Lamp1-Yellow
        Rectangle (31,68 213x19), "Safety Sick Flexi Soft"
    Rectangle (510,791 237x20), "Dispositivos Safety"
    Rectangle (510,809 237x20), "XTIO[1] - 8 entradas e 4 Saídas"
    Rectangle (547,829 204x19), "I1-I2 - Botão de Emergência"
    Lamp1 (507,829 20x20), variable: I2, style: Lamp-Lamp1-Yellow
    Lamp1 (527,829 20x20), variable: I2, style: Lamp-Lamp1-Yellow
    Rectangle (547,849 204x19), "I3-I4 - Botão de Emergência"
    Lamp1 (507,849 20x20), variable: I2, style: Lamp-Lamp1-Yellow
    Lamp1 (527,849 20x20), variable: I2, style: Lamp-Lamp1-Yellow
    Lamp1 (507,869 20x20), variable: I2, style: Lamp-Lamp1-Yellow
    Rectangle (547,869 204x19), "I3-I4 - Botão de Emergência"
    Lamp1 (527,869 20x20), variable: I2, style: Lamp-Lamp1-Yellow
    Lamp1 (507,889 20x20), variable: I2, style: Lamp-Lamp1-Yellow
    Rectangle (547,889 204x19), "I3-I4 - Botão de Emergência"
    Lamp1 (527,889 20x20), variable: I2, style: Lamp-Lamp1-Yellow
    Lamp1 (507,909 20x20), variable: I2, style: Lamp-Lamp1-Yellow
    Rectangle (547,909 204x19), "Q1-Q2 - Servo 1"
    Lamp1 (527,909 20x20), variable: I2, style: Lamp-Lamp1-Yellow
    Lamp1 (507,929 20x20), variable: I2, style: Lamp-Lamp1-Yellow
    Rectangle (547,929 204x19), "Q3-Q4 - Servo 2"
    Lamp1 (527,929 20x20), variable: I2, style: Lamp-Lamp1-Yellow
    Rectangle (510,952 237x20), "XTIO[2] - 8 entradas e 4 Saídas"
    Rectangle (547,972 204x19), "I1-I2 - Cortina de Luz"
    Lamp1 (507,972 20x20), variable: I2, style: Lamp-Lamp1-Yellow
    Lamp1 (527,972 20x20), variable: I2, style: Lamp-Lamp1-Yellow
    Rectangle (547,992 204x19), "I3-I4 - Sensor Porta"
    Lamp1 (507,992 20x20), variable: I2, style: Lamp-Lamp1-Yellow
    Lamp1 (527,992 20x20), variable: I2, style: Lamp-Lamp1-Yellow
    Lamp1 (507,1012 20x20), variable: I2, style: Lamp-Lamp1-Yellow
    Rectangle (547,1012 204x19), "I3-I4 - Sensor Porta"
    Lamp1 (527,1012 20x20), variable: I2, style: Lamp-Lamp1-Yellow
    Lamp1 (507,1032 20x20), variable: I2, style: Lamp-Lamp1-Yellow
    Rectangle (547,1032 204x19), "I3-I4 - Sensor Porta"
    Lamp1 (527,1032 20x20), variable: I2, style: Lamp-Lamp1-Yellow
    Lamp1 (507,1052 20x20), variable: I2, style: Lamp-Lamp1-Yellow
    Rectangle (547,1052 204x19), "Q1-Q2 - Motor"
    Lamp1 (527,1052 20x20), variable: I2, style: Lamp-Lamp1-Yellow
    Lamp1 (507,1072 20x20), variable: I2, style: Lamp-Lamp1-Yellow
    Rectangle (547,1072 204x19), "Q3-Q4 - Motor"
    Lamp1 (527,1072 20x20), variable: I2, style: Lamp-Lamp1-Yellow
    Rectangle (507,1094 237x20), "XTIO[3] - 8 entradas e 4 Saídas"
    Rectangle (544,1114 204x19), "I1-I2 - Sensor Porta"
    Lamp1 (504,1114 20x20), variable: I2, style: Lamp-Lamp1-Yellow
    Lamp1 (524,1114 20x20), variable: I2, style: Lamp-Lamp1-Yellow
    Rectangle (544,1134 204x19), "I3-I4 - Sensor Porta"
    Lamp1 (504,1134 20x20), variable: I2, style: Lamp-Lamp1-Yellow
    Lamp1 (524,1134 20x20), variable: I2, style: Lamp-Lamp1-Yellow
    Lamp1 (504,1154 20x20), variable: I2, style: Lamp-Lamp1-Yellow
    Rectangle (544,1154 204x19), "I3-I4 - Sensor Porta"
    Lamp1 (524,1154 20x20), variable: I2, style: Lamp-Lamp1-Yellow
    Lamp1 (504,1174 20x20), variable: I2, style: Lamp-Lamp1-Yellow
    Rectangle (544,1174 204x19), "I3-I4 - Sensor Porta"
    Lamp1 (524,1174 20x20), variable: I2, style: Lamp-Lamp1-Yellow
    Lamp1 (504,1194 20x20), variable: I2, style: Lamp-Lamp1-Yellow
    Rectangle (544,1194 204x19), "Q1-Q2 - Robo Yaskawa GP7"
    Lamp1 (524,1194 20x20), variable: I2, style: Lamp-Lamp1-Yellow
    Lamp1 (504,1214 20x20), variable: I2, style: Lamp-Lamp1-Yellow
    Rectangle (544,1214 204x19), "Q3-Q4 - Reserva"
    Lamp1 (524,1214 20x20), variable: I2, style: Lamp-Lamp1-Yellow
    Button (15,1315 175x45), "RECEITAS"
        OnMouseClick: change screen: Tela_Receita
    Button (375,1315 175x45), "MOV. MANUAIS"
        OnMouseClick: change screen: Tela_Manual_1
    Button (195,1315 175x45), "PRODUÇÃO"
        OnMouseClick: change screen: Tela_Producao
END_VISUALIZATION
